{attribute 'GeneratedUsingTerminal: EK1100-0000-0018'}
{attribute addProperty BoxType "EK1100-0000-0018"}
{attribute addProperty Id "Beckhoff_EL30xxEK1122Beckhoff_EL30xxEK1122_83BFF9012A_0001_EL3001_0000_0016EL3001_4F06975421A_0002_EL3001_0000_0017EL3001_1300E0B121A_0003_EL3001_0000_0018EL3001_1300E0B121A_0004_EL3001_0000_0019EL3001_1300E0B121A_0005_EL3001_0000_0020EL3001_1300E0B121A_0006_EL3001_0000_0021EL3001_1300E0B121A_0007_EL3002_0000_0016EL3002_FE294BE330A_0008_EL3002_0000_0017EL3002_620EF68730A_0009_EL3002_0000_0018EL3002_620EF68730A_0010_EL3002_0000_0019EL3002_620EF68730A_0011_EL3002_0000_0020EL3002_620EF68730A_0012_EL3002_0000_0021EL3002_620EF68730A_0013_EL3004_0000_0016EL3004_B1E8798348A_0014_EL3004_0000_0017EL3004_9DDA7BAE48A_0015_EL3004_0000_0018EL3004_9DDA7BAE48A_0016_EL3004_0000_0019EL3004_9DDA7BAE48A_0017_EL3004_0000_0020EL3004_9DDA7BAE48A_0018_EL3004_0000_0021EL3004_9DDA7BAE48A_0019_EL3008_0000_0016EL3008_DA7971F784A_0020_EL3008_0000_0017EL3008_085DE50284A_0021_EL3008_0000_0018EL3008_085DE50284A_0022_EL3008_0000_0019EL3008_085DE50284A_0023_EL3008_0000_0020EL3008_085DE50284A_0024_EL3008_0000_0021EL3008_085DE50284A_0025_EL3011_0000_0016EL3011_1300E0B121A_0026_EL3011_0000_0017EL3011_1300E0B121A_0027_EL3011_0000_0018EL3011_1300E0B121A_0028_EL3011_0000_0019EL3011_1300E0B121A_0029_EL3011_0000_0020EL3011_1300E0B121A_0030_EL3012_0000_0016EL3012_620EF68730A_0031_EL3012_0000_0017EL3012_620EF68730A_0032_EL3012_0000_0018EL3012_620EF68730A_0033_EL3012_0000_0019EL3012_620EF68730A_0034_EL3012_0000_0020EL3012_620EF68730A_0035_EL3014_0000_0016EL3014_9DDA7BAE48A_0036_EL3014_0000_0017EL3014_9DDA7BAE48A_0037_EL3014_0000_0018EL3014_9DDA7BAE48A_0038_EL3014_0000_0019EL3014_9DDA7BAE48A_0039_EL3021_0000_0016EL3021_1300E0B121A_0040_EL3021_0000_0017EL3021_1300E0B121A_0041_EL3021_0000_0018EL3021_1300E0B121A_0042_EL3021_0000_0019EL3021_1300E0B121A_0043_EL3021_0000_0020EL3021_1300E0B121A_0044_EL3022_0000_0016EL3022_620EF68730A_0045_EL3022_0000_0017EL3022_620EF68730A_0046_EL3022_0000_0018EL3022_620EF68730A_0047_EL3022_0000_0019EL3022_620EF68730A_0048_EL3022_0000_0020EL3022_620EF68730A_0049_EL3024_0000_0016EL3024_9DDA7BAE48A_0050_EL3024_0000_0017EL3024_9DDA7BAE48A_0051_EL3024_0000_0018EL3024_9DDA7BAE48A_0052_EL3024_0000_0019EL3024_9DDA7BAE48A_0053_EL3041_0000_0016EL3041_4F06975421A_0054_EL3041_0000_0017EL3041_1300E0B121A_0055_EL3041_0000_0018EL3041_1300E0B121A_0056_EL3041_0000_0019EL3041_1300E0B121A_0057_EL3041_0000_0020EL3041_1300E0B121A_0058_EL3042_0000_0016EL3042_FE294BE330A_0059_EL3042_0000_0017EL3042_620EF68730A_0060_EL3042_0000_0018EL3042_620EF68730A_0061_EL3042_0000_0019EL3042_620EF68730A_0062_EL3042_0000_0020EL3042_620EF68730A_0063_EL3042_0017_0016EL3042_FE294BE330A_0064_EL3042_0017_0017EL3042_620EF68730A_0065_EL3042_0017_0018EL3042_620EF68730A_0066_EL3042_0017_0019EL3042_620EF68730A_0067_EL3042_0017_0020EL3042_620EF68730A_0068_EL3042_0017_0021EL3042_620EF68730A_0069_EL3044_0000_0016EL3044_B1E8798348A_0070_EL3044_0000_0017EL3044_9DDA7BAE48A_0071_EL3044_0000_0018EL3044_9DDA7BAE48A_0072_EL3044_0000_0019EL3044_9DDA7BAE48A_0073_EL3044_0000_0020EL3044_9DDA7BAE48A_0074_EL3048_0000_0016EL3048_DA7971F784A_0075_EL3048_0000_0017EL3048_085DE50284A_0076_EL3048_0000_0018EL3048_085DE50284A_0077_EL3048_0000_0019EL3048_085DE50284A_0078_EL3048_0000_0020EL3048_085DE50284A_0079_EL3051_0000_0016EL3051_4F06975421A_0080_EL3051_0000_0017EL3051_1300E0B121A_0081_EL3051_0000_0018EL3051_1300E0B121A_0082_EL3051_0000_0019EL3051_1300E0B121A_0083_EL3051_0000_0020EL3051_1300E0B121A_0084_EL3052_0000_0016EL3052_FE294BE330A_0085_EL3052_0000_0017EL3052_620EF68730A_0086_EL3052_0000_0018EL3052_620EF68730A_0087_EL3052_0000_0019EL3052_620EF68730A_0088_EL3052_0000_0020EL3052_620EF68730A_0089_EL3054_0000_0016EL3054_B1E8798348A_0090_EL3054_0000_0017EL3054_9DDA7BAE48A_0091_EL3054_0000_0018EL3054_9DDA7BAE48A_0092_EL3054_0000_0019EL3054_9DDA7BAE48A_0093_EL3054_0000_0020EL3054_9DDA7BAE48A_0094_EL3058_0000_0016EL3058_DA7971F784A_0095_EL3058_0000_0017EL3058_085DE50284A_0096_EL3058_0000_0018EL3058_085DE50284A_0097_EL3058_0000_0019EL3058_085DE50284A_0098_EL3058_0000_0020EL3058_085DE50284A_0099_EL3061_0000_0016EL3061_4F06975421A_0100_EL3061_0000_0017EL3061_1300E0B121A_0101_EL3061_0000_0018EL3061_1300E0B121A_0102_EL3061_0000_0019EL3061_1300E0B121A_0103_EL3061_0000_0020EL3061_1300E0B121A_0104_EL3062_0000_0016EL3062_FE294BE330A_0105_EL3062_0000_0017EL3062_620EF68730A_0106_EL3062_0000_0018EL3062_620EF68730A_0107_EL3062_0000_0019EL3062_620EF68730A_0108_EL3062_0000_0020EL3062_620EF68730A_0109_EL3062_0015_0016EL3062_620EF68730A_0110_EL3062_0030_0016EL3062_FE294BE330A_0111_EL3062_0030_0017EL3062_620EF68730A_0112_EL3062_0030_0018EL3062_620EF68730A_0113_EL3062_0030_0019EL3062_620EF68730A_0114_EL3062_0030_0020EL3062_620EF68730A_0115_EL3062_0030_0021EL3062_620EF68730A_0116_EL3064_0000_0016EL3064_B1E8798348A_0117_EL3064_0000_0017EL3064_9DDA7BAE48A_0118_EL3064_0000_0018EL3064_9DDA7BAE48A_0119_EL3064_0000_0019EL3064_9DDA7BAE48A_0120_EL3064_0000_0020EL3064_9DDA7BAE48A_0121_EL3068_0000_0016EL3068_DA7971F784A_0122_EL3068_0000_0017EL3068_085DE50284A_0123_EL3068_0000_0018EL3068_085DE50284A_0124_EL3068_0000_0019EL3068_085DE50284A_0125_EL3068_0000_0020EL3068_085DE50284"}
{attribute addProperty CRC "2209379809"}
{attribute addProperty Size "5129"}
TYPE Beckhoff_EL30xx_83B075E1 EXTENDS EK1100_AB5A9467 :
STRUCT
	{attribute addProperty Name "Beckhoff_EL30xxEK1122"}
	Beckhoff_EL30xxEK1122 : Beckhoff_EL30xxEK1122_83BFF901;
	{attribute addProperty Name "A_0001_EL3001_0000_0016"}
	A_0001_EL3001_0000_0016 : EL3001_4F069754;
	{attribute addProperty Name "A_0002_EL3001_0000_0017"}
	A_0002_EL3001_0000_0017 : EL3001_1300E0B1;
	{attribute addProperty Name "A_0003_EL3001_0000_0018"}
	A_0003_EL3001_0000_0018 : EL3001_1300E0B1;
	{attribute addProperty Name "A_0004_EL3001_0000_0019"}
	A_0004_EL3001_0000_0019 : EL3001_1300E0B1;
	{attribute addProperty Name "A_0005_EL3001_0000_0020"}
	A_0005_EL3001_0000_0020 : EL3001_1300E0B1;
	{attribute addProperty Name "A_0006_EL3001_0000_0021"}
	A_0006_EL3001_0000_0021 : EL3001_1300E0B1;
	{attribute addProperty Name "A_0007_EL3002_0000_0016"}
	A_0007_EL3002_0000_0016 : EL3002_FE294BE3;
	{attribute addProperty Name "A_0008_EL3002_0000_0017"}
	A_0008_EL3002_0000_0017 : EL3002_620EF687;
	{attribute addProperty Name "A_0009_EL3002_0000_0018"}
	A_0009_EL3002_0000_0018 : EL3002_620EF687;
	{attribute addProperty Name "A_0010_EL3002_0000_0019"}
	A_0010_EL3002_0000_0019 : EL3002_620EF687;
	{attribute addProperty Name "A_0011_EL3002_0000_0020"}
	A_0011_EL3002_0000_0020 : EL3002_620EF687;
	{attribute addProperty Name "A_0012_EL3002_0000_0021"}
	A_0012_EL3002_0000_0021 : EL3002_620EF687;
	{attribute addProperty Name "A_0013_EL3004_0000_0016"}
	A_0013_EL3004_0000_0016 : EL3004_B1E87983;
	{attribute addProperty Name "A_0014_EL3004_0000_0017"}
	A_0014_EL3004_0000_0017 : EL3004_9DDA7BAE;
	{attribute addProperty Name "A_0015_EL3004_0000_0018"}
	A_0015_EL3004_0000_0018 : EL3004_9DDA7BAE;
	{attribute addProperty Name "A_0016_EL3004_0000_0019"}
	A_0016_EL3004_0000_0019 : EL3004_9DDA7BAE;
	{attribute addProperty Name "A_0017_EL3004_0000_0020"}
	A_0017_EL3004_0000_0020 : EL3004_9DDA7BAE;
	{attribute addProperty Name "A_0018_EL3004_0000_0021"}
	A_0018_EL3004_0000_0021 : EL3004_9DDA7BAE;
	{attribute addProperty Name "A_0019_EL3008_0000_0016"}
	A_0019_EL3008_0000_0016 : EL3008_DA7971F7;
	{attribute addProperty Name "A_0020_EL3008_0000_0017"}
	A_0020_EL3008_0000_0017 : EL3008_085DE502;
	{attribute addProperty Name "A_0021_EL3008_0000_0018"}
	A_0021_EL3008_0000_0018 : EL3008_085DE502;
	{attribute addProperty Name "A_0022_EL3008_0000_0019"}
	A_0022_EL3008_0000_0019 : EL3008_085DE502;
	{attribute addProperty Name "A_0023_EL3008_0000_0020"}
	A_0023_EL3008_0000_0020 : EL3008_085DE502;
	{attribute addProperty Name "A_0024_EL3008_0000_0021"}
	A_0024_EL3008_0000_0021 : EL3008_085DE502;
	{attribute addProperty Name "A_0025_EL3011_0000_0016"}
	A_0025_EL3011_0000_0016 : EL3011_1300E0B1;
	{attribute addProperty Name "A_0026_EL3011_0000_0017"}
	A_0026_EL3011_0000_0017 : EL3011_1300E0B1;
	{attribute addProperty Name "A_0027_EL3011_0000_0018"}
	A_0027_EL3011_0000_0018 : EL3011_1300E0B1;
	{attribute addProperty Name "A_0028_EL3011_0000_0019"}
	A_0028_EL3011_0000_0019 : EL3011_1300E0B1;
	{attribute addProperty Name "A_0029_EL3011_0000_0020"}
	A_0029_EL3011_0000_0020 : EL3011_1300E0B1;
	{attribute addProperty Name "A_0030_EL3012_0000_0016"}
	A_0030_EL3012_0000_0016 : EL3012_620EF687;
	{attribute addProperty Name "A_0031_EL3012_0000_0017"}
	A_0031_EL3012_0000_0017 : EL3012_620EF687;
	{attribute addProperty Name "A_0032_EL3012_0000_0018"}
	A_0032_EL3012_0000_0018 : EL3012_620EF687;
	{attribute addProperty Name "A_0033_EL3012_0000_0019"}
	A_0033_EL3012_0000_0019 : EL3012_620EF687;
	{attribute addProperty Name "A_0034_EL3012_0000_0020"}
	A_0034_EL3012_0000_0020 : EL3012_620EF687;
	{attribute addProperty Name "A_0035_EL3014_0000_0016"}
	A_0035_EL3014_0000_0016 : EL3014_9DDA7BAE;
	{attribute addProperty Name "A_0036_EL3014_0000_0017"}
	A_0036_EL3014_0000_0017 : EL3014_9DDA7BAE;
	{attribute addProperty Name "A_0037_EL3014_0000_0018"}
	A_0037_EL3014_0000_0018 : EL3014_9DDA7BAE;
	{attribute addProperty Name "A_0038_EL3014_0000_0019"}
	A_0038_EL3014_0000_0019 : EL3014_9DDA7BAE;
	{attribute addProperty Name "A_0039_EL3021_0000_0016"}
	A_0039_EL3021_0000_0016 : EL3021_1300E0B1;
	{attribute addProperty Name "A_0040_EL3021_0000_0017"}
	A_0040_EL3021_0000_0017 : EL3021_1300E0B1;
	{attribute addProperty Name "A_0041_EL3021_0000_0018"}
	A_0041_EL3021_0000_0018 : EL3021_1300E0B1;
	{attribute addProperty Name "A_0042_EL3021_0000_0019"}
	A_0042_EL3021_0000_0019 : EL3021_1300E0B1;
	{attribute addProperty Name "A_0043_EL3021_0000_0020"}
	A_0043_EL3021_0000_0020 : EL3021_1300E0B1;
	{attribute addProperty Name "A_0044_EL3022_0000_0016"}
	A_0044_EL3022_0000_0016 : EL3022_620EF687;
	{attribute addProperty Name "A_0045_EL3022_0000_0017"}
	A_0045_EL3022_0000_0017 : EL3022_620EF687;
	{attribute addProperty Name "A_0046_EL3022_0000_0018"}
	A_0046_EL3022_0000_0018 : EL3022_620EF687;
	{attribute addProperty Name "A_0047_EL3022_0000_0019"}
	A_0047_EL3022_0000_0019 : EL3022_620EF687;
	{attribute addProperty Name "A_0048_EL3022_0000_0020"}
	A_0048_EL3022_0000_0020 : EL3022_620EF687;
	{attribute addProperty Name "A_0049_EL3024_0000_0016"}
	A_0049_EL3024_0000_0016 : EL3024_9DDA7BAE;
	{attribute addProperty Name "A_0050_EL3024_0000_0017"}
	A_0050_EL3024_0000_0017 : EL3024_9DDA7BAE;
	{attribute addProperty Name "A_0051_EL3024_0000_0018"}
	A_0051_EL3024_0000_0018 : EL3024_9DDA7BAE;
	{attribute addProperty Name "A_0052_EL3024_0000_0019"}
	A_0052_EL3024_0000_0019 : EL3024_9DDA7BAE;
	{attribute addProperty Name "A_0053_EL3041_0000_0016"}
	A_0053_EL3041_0000_0016 : EL3041_4F069754;
	{attribute addProperty Name "A_0054_EL3041_0000_0017"}
	A_0054_EL3041_0000_0017 : EL3041_1300E0B1;
	{attribute addProperty Name "A_0055_EL3041_0000_0018"}
	A_0055_EL3041_0000_0018 : EL3041_1300E0B1;
	{attribute addProperty Name "A_0056_EL3041_0000_0019"}
	A_0056_EL3041_0000_0019 : EL3041_1300E0B1;
	{attribute addProperty Name "A_0057_EL3041_0000_0020"}
	A_0057_EL3041_0000_0020 : EL3041_1300E0B1;
	{attribute addProperty Name "A_0058_EL3042_0000_0016"}
	A_0058_EL3042_0000_0016 : EL3042_FE294BE3;
	{attribute addProperty Name "A_0059_EL3042_0000_0017"}
	A_0059_EL3042_0000_0017 : EL3042_620EF687;
	{attribute addProperty Name "A_0060_EL3042_0000_0018"}
	A_0060_EL3042_0000_0018 : EL3042_620EF687;
	{attribute addProperty Name "A_0061_EL3042_0000_0019"}
	A_0061_EL3042_0000_0019 : EL3042_620EF687;
	{attribute addProperty Name "A_0062_EL3042_0000_0020"}
	A_0062_EL3042_0000_0020 : EL3042_620EF687;
	{attribute addProperty Name "A_0063_EL3042_0017_0016"}
	A_0063_EL3042_0017_0016 : EL3042_FE294BE3;
	{attribute addProperty Name "A_0064_EL3042_0017_0017"}
	A_0064_EL3042_0017_0017 : EL3042_620EF687;
	{attribute addProperty Name "A_0065_EL3042_0017_0018"}
	A_0065_EL3042_0017_0018 : EL3042_620EF687;
	{attribute addProperty Name "A_0066_EL3042_0017_0019"}
	A_0066_EL3042_0017_0019 : EL3042_620EF687;
	{attribute addProperty Name "A_0067_EL3042_0017_0020"}
	A_0067_EL3042_0017_0020 : EL3042_620EF687;
	{attribute addProperty Name "A_0068_EL3042_0017_0021"}
	A_0068_EL3042_0017_0021 : EL3042_620EF687;
	{attribute addProperty Name "A_0069_EL3044_0000_0016"}
	A_0069_EL3044_0000_0016 : EL3044_B1E87983;
	{attribute addProperty Name "A_0070_EL3044_0000_0017"}
	A_0070_EL3044_0000_0017 : EL3044_9DDA7BAE;
	{attribute addProperty Name "A_0071_EL3044_0000_0018"}
	A_0071_EL3044_0000_0018 : EL3044_9DDA7BAE;
	{attribute addProperty Name "A_0072_EL3044_0000_0019"}
	A_0072_EL3044_0000_0019 : EL3044_9DDA7BAE;
	{attribute addProperty Name "A_0073_EL3044_0000_0020"}
	A_0073_EL3044_0000_0020 : EL3044_9DDA7BAE;
	{attribute addProperty Name "A_0074_EL3048_0000_0016"}
	A_0074_EL3048_0000_0016 : EL3048_DA7971F7;
	{attribute addProperty Name "A_0075_EL3048_0000_0017"}
	A_0075_EL3048_0000_0017 : EL3048_085DE502;
	{attribute addProperty Name "A_0076_EL3048_0000_0018"}
	A_0076_EL3048_0000_0018 : EL3048_085DE502;
	{attribute addProperty Name "A_0077_EL3048_0000_0019"}
	A_0077_EL3048_0000_0019 : EL3048_085DE502;
	{attribute addProperty Name "A_0078_EL3048_0000_0020"}
	A_0078_EL3048_0000_0020 : EL3048_085DE502;
	{attribute addProperty Name "A_0079_EL3051_0000_0016"}
	A_0079_EL3051_0000_0016 : EL3051_4F069754;
	{attribute addProperty Name "A_0080_EL3051_0000_0017"}
	A_0080_EL3051_0000_0017 : EL3051_1300E0B1;
	{attribute addProperty Name "A_0081_EL3051_0000_0018"}
	A_0081_EL3051_0000_0018 : EL3051_1300E0B1;
	{attribute addProperty Name "A_0082_EL3051_0000_0019"}
	A_0082_EL3051_0000_0019 : EL3051_1300E0B1;
	{attribute addProperty Name "A_0083_EL3051_0000_0020"}
	A_0083_EL3051_0000_0020 : EL3051_1300E0B1;
	{attribute addProperty Name "A_0084_EL3052_0000_0016"}
	A_0084_EL3052_0000_0016 : EL3052_FE294BE3;
	{attribute addProperty Name "A_0085_EL3052_0000_0017"}
	A_0085_EL3052_0000_0017 : EL3052_620EF687;
	{attribute addProperty Name "A_0086_EL3052_0000_0018"}
	A_0086_EL3052_0000_0018 : EL3052_620EF687;
	{attribute addProperty Name "A_0087_EL3052_0000_0019"}
	A_0087_EL3052_0000_0019 : EL3052_620EF687;
	{attribute addProperty Name "A_0088_EL3052_0000_0020"}
	A_0088_EL3052_0000_0020 : EL3052_620EF687;
	{attribute addProperty Name "A_0089_EL3054_0000_0016"}
	A_0089_EL3054_0000_0016 : EL3054_B1E87983;
	{attribute addProperty Name "A_0090_EL3054_0000_0017"}
	A_0090_EL3054_0000_0017 : EL3054_9DDA7BAE;
	{attribute addProperty Name "A_0091_EL3054_0000_0018"}
	A_0091_EL3054_0000_0018 : EL3054_9DDA7BAE;
	{attribute addProperty Name "A_0092_EL3054_0000_0019"}
	A_0092_EL3054_0000_0019 : EL3054_9DDA7BAE;
	{attribute addProperty Name "A_0093_EL3054_0000_0020"}
	A_0093_EL3054_0000_0020 : EL3054_9DDA7BAE;
	{attribute addProperty Name "A_0094_EL3058_0000_0016"}
	A_0094_EL3058_0000_0016 : EL3058_DA7971F7;
	{attribute addProperty Name "A_0095_EL3058_0000_0017"}
	A_0095_EL3058_0000_0017 : EL3058_085DE502;
	{attribute addProperty Name "A_0096_EL3058_0000_0018"}
	A_0096_EL3058_0000_0018 : EL3058_085DE502;
	{attribute addProperty Name "A_0097_EL3058_0000_0019"}
	A_0097_EL3058_0000_0019 : EL3058_085DE502;
	{attribute addProperty Name "A_0098_EL3058_0000_0020"}
	A_0098_EL3058_0000_0020 : EL3058_085DE502;
	{attribute addProperty Name "A_0099_EL3061_0000_0016"}
	A_0099_EL3061_0000_0016 : EL3061_4F069754;
	{attribute addProperty Name "A_0100_EL3061_0000_0017"}
	A_0100_EL3061_0000_0017 : EL3061_1300E0B1;
	{attribute addProperty Name "A_0101_EL3061_0000_0018"}
	A_0101_EL3061_0000_0018 : EL3061_1300E0B1;
	{attribute addProperty Name "A_0102_EL3061_0000_0019"}
	A_0102_EL3061_0000_0019 : EL3061_1300E0B1;
	{attribute addProperty Name "A_0103_EL3061_0000_0020"}
	A_0103_EL3061_0000_0020 : EL3061_1300E0B1;
	{attribute addProperty Name "A_0104_EL3062_0000_0016"}
	A_0104_EL3062_0000_0016 : EL3062_FE294BE3;
	{attribute addProperty Name "A_0105_EL3062_0000_0017"}
	A_0105_EL3062_0000_0017 : EL3062_620EF687;
	{attribute addProperty Name "A_0106_EL3062_0000_0018"}
	A_0106_EL3062_0000_0018 : EL3062_620EF687;
	{attribute addProperty Name "A_0107_EL3062_0000_0019"}
	A_0107_EL3062_0000_0019 : EL3062_620EF687;
	{attribute addProperty Name "A_0108_EL3062_0000_0020"}
	A_0108_EL3062_0000_0020 : EL3062_620EF687;
	{attribute addProperty Name "A_0109_EL3062_0015_0016"}
	A_0109_EL3062_0015_0016 : EL3062_620EF687;
	{attribute addProperty Name "A_0110_EL3062_0030_0016"}
	A_0110_EL3062_0030_0016 : EL3062_FE294BE3;
	{attribute addProperty Name "A_0111_EL3062_0030_0017"}
	A_0111_EL3062_0030_0017 : EL3062_620EF687;
	{attribute addProperty Name "A_0112_EL3062_0030_0018"}
	A_0112_EL3062_0030_0018 : EL3062_620EF687;
	{attribute addProperty Name "A_0113_EL3062_0030_0019"}
	A_0113_EL3062_0030_0019 : EL3062_620EF687;
	{attribute addProperty Name "A_0114_EL3062_0030_0020"}
	A_0114_EL3062_0030_0020 : EL3062_620EF687;
	{attribute addProperty Name "A_0115_EL3062_0030_0021"}
	A_0115_EL3062_0030_0021 : EL3062_620EF687;
	{attribute addProperty Name "A_0116_EL3064_0000_0016"}
	A_0116_EL3064_0000_0016 : EL3064_B1E87983;
	{attribute addProperty Name "A_0117_EL3064_0000_0017"}
	A_0117_EL3064_0000_0017 : EL3064_9DDA7BAE;
	{attribute addProperty Name "A_0118_EL3064_0000_0018"}
	A_0118_EL3064_0000_0018 : EL3064_9DDA7BAE;
	{attribute addProperty Name "A_0119_EL3064_0000_0019"}
	A_0119_EL3064_0000_0019 : EL3064_9DDA7BAE;
	{attribute addProperty Name "A_0120_EL3064_0000_0020"}
	A_0120_EL3064_0000_0020 : EL3064_9DDA7BAE;
	{attribute addProperty Name "A_0121_EL3068_0000_0016"}
	A_0121_EL3068_0000_0016 : EL3068_DA7971F7;
	{attribute addProperty Name "A_0122_EL3068_0000_0017"}
	A_0122_EL3068_0000_0017 : EL3068_085DE502;
	{attribute addProperty Name "A_0123_EL3068_0000_0018"}
	A_0123_EL3068_0000_0018 : EL3068_085DE502;
	{attribute addProperty Name "A_0124_EL3068_0000_0019"}
	A_0124_EL3068_0000_0019 : EL3068_085DE502;
	{attribute addProperty Name "A_0125_EL3068_0000_0020"}
	A_0125_EL3068_0000_0020 : EL3068_085DE502;
END_STRUCT
END_TYPE

(* stored: Version 1.2.0.0, ProductVersion 3.1.4024.9
   DUT Beckhoff_EL30xx_83B075E1: Id {c4baf300-e24e-4432-8295-547775a27453} *)
